TYPE ST_AutomaticExtractionParameters :
STRUCT
	fillingTime : DINT;
	pumpSetpointWaitTime : DINT;
	pumpOnTime	: DINT;
	controlValveOpeningValue : DINT;
END_STRUCT
END_TYPE

(* stored: Version 1.1.0.1, ProductVersion 3.1.4024.9
   DUT ST_AutomaticExtractionParameters: Id {09f81920-6f18-4345-a1f6-809bcfa5979e} *)
